{attribute 'qualified_only'}
{attribute 'strict'}
{attribute 'to_string'}
TYPE E_MOVER_CTRL :
(
  MOVER_NULL,               // initial value at startup, used for change of order or retrigger
  MOVER_ENABLE,             // sets MC_Power.Enable
  MOVER_DISABLE,            // removes MC_Power.Enable
  MOVER_MOVE_TO_POS,        // modulo absolute positioning with MC_MoveAbsolute, InTargetPosition check
  MOVER_MOVE_TO_POS_CA,     // modulo absolute positioning with MC_MoveAbsoluteCA, InTargetPosition check
  MOVER_SEND_TO_POS_CA,     // modulo absolute positioning with MC_MoveAbsoluteCA, done after moving ReleaseDistance
  MOVER_HALT,               // halts mover; by use of MC_Halt mover is set passive in CA group
  MOVER_GEAR_IN,            // GearIn for mover in standstill

  MOVER_GEAR_IN_POS_CA,     // GearInPosCA of mover; when FB_GearInPosCa is InSync --> order is done; check SyncDistance yourself and release mover with e_mover_order.mover_SendToPos
  MOVER_GEAR_OUT,           // gear out for mover
  MOVER_RESET,              // MC_RESET for mover
  MOVER_INFO                // used to display MoverInfo in ST_MOVER_SELECTOR_STATE.Info
)UINT;
END_TYPE

(* stored: Version 1.1.0.1, ProductVersion 3.1.4026.20
   DUT E_MOVER_CTRL: Id {7c09cc4d-2d74-4d3f-842f-b3137d2f85c0} *)
